FUNCTION_BLOCK ExampleFlashingLamp_Composition IMPLEMENTS I_Instance, I_CyclicInstance
VAR
	instance : Instance;
	taskMembership : AutomaticGlobalInstanceMembership(THIS^);
	_cyclicCallback : CyclicCallback(THIS^);

	tick : ton;
	tock : ton;
END_VAR

// To make an object cyclic called via composition then you must implement I_Instance and I_CyclicInstance
// and also contain a GlobalInstanceMembership.
//
// I_Instance 
// This can be done by creating variable of type Instance and linking your own .Namespace 
// and .ShareNamespaceWith() with it.  
//
// I_CyclicInstance 
// You must make a callback by the name of CyclicInstanceCallback which will be auto subscribed by the task.
// The premade CyclicCallback

METHOD CyclicCall
VAR_INPUT
END_VAR
tick(in:=NOT tock.Q,pt:=T#1S);
tock(in:=tick.Q,pt:=T#1S);
END_METHOD

PROPERTY PUBLIC CyclicInstanceCallback : I_Callback
GET
CyclicInstanceCallback := _cyclicCallback;
END_GET
END_PROPERTY

PROPERTY PUBLIC NameSpace : STRING
GET
Namespace := instance.Namespace;
END_GET
END_PROPERTY

PROPERTY PUBLIC Output : BOOL
GET
Output := tick.Q;
END_GET
END_PROPERTY

METHOD PUBLIC SharesNamespaceWith : BOOL
VAR_INPUT
	OtherInstance : I_Instance;
END_VAR
SharesNamespaceWith := instance.SharesNamespaceWith(OtherInstance);
END_METHOD

END_FUNCTION_BLOCK

(* stored: Version 1.1.0.1, ProductVersion 3.1.4024.11
   POU ExampleFlashingLamp_Composition: Id {6c346b92-d0ba-425a-8541-d59d40052e70}, SpecialFunc None
   Folder Required for I_CyclicInstance: Id {085084e1-28b8-49b0-a33b-c32bd6c2ca30}
   Folder Required for I_Instance: Id {44b1aaf6-8874-4606-b8bd-311fdf0035ed}
   Method CyclicCall: Id {7d561706-baad-496a-b32c-52968374d31e}
   Property CyclicInstanceCallback: Id {3a37ff4e-49ad-4396-846e-88601200eb49}
   Get Get: Id {f4fa7f7a-4187-459d-bbd4-542d29aa4452}
   Property NameSpace: Id {303c425b-90e1-4160-9417-10a402bf031e}
   Get Get: Id {371df91b-4908-40bd-af7c-1ba9ee414ab6}
   Property Output: Id {3cd6e915-b5bb-4734-b503-20e7a939da3e}
   Get Get: Id {0ca7be68-adbb-43ce-a354-07885449c9ef}
   Method SharesNamespaceWith: Id {871d87d6-9233-44b7-864b-7ceeb3ada5a0} *)
